TYPE ST_GCSingleProcessStageTiming :
STRUCT
	StartUtc : STRING(20);
	EndUtc : STRING(20);
	TargetTime : TIME;
	ActualTime : TIME;
	Timeout : TIME;
	Completed : BOOL;
	TimedOut : BOOL;
END_STRUCT
END_TYPE

(* stored: Version 1.1.0.1, ProductVersion 3.1.4026.18
   DUT ST_GCSingleProcessStageTiming: Id {c553a379-09a6-4064-a509-cb15e95859d3} *)
